(*
Récupère la Config de AppConfig
Démarre HardwareManager
Todo : Démarre la Bdd
Todo : Démarre le monitoring
*)

FUNCTION_BLOCK HardwareControl
VAR_INPUT
END_VAR
VAR_OUTPUT
END_VAR
VAR
	{region "manage file" }	
	{attribute 'OPC.UA.DA' := '0'}	
	_xml : TXml;	
	{attribute 'hide'}
	_filePath : T_MaxString := Const.APP_CONFIG_FILE_PATH; 
	{attribute 'hide'}  			
    _xPath : T_MaxString := Const.APP_CONFIG_XPATH; 
	{endregion}		
		
	{attribute 'hide'}  
	_loadConfigDone : BOOL;
	{attribute 'OPC.UA.DA' := '0'}
	_initialized : BOOL;
	{attribute 'OPC.UA.DA' := '0'}
	_initializedError : BOOL;	
	{attribute 'OPC.UA.DA' := '0'}
	_message : StringBuilder;
	{attribute 'OPC.UA.DA' := '0'}
	_logger : Logger;
	
	autoBoot : BOOL := TRUE;
	
	HardwareManager : HardwareManager;	
END_VAR

IF autoBoot THEN
	InitHardware();
END_IF

ACTION AppDeserialize:
_xml(FilePath := _filePath, XPath := _xPath, 
	 AddHeaderNodeXml := ADR(GlobalConfig.AppConfig), 
	 SizeOfHeaderNodeXml := SIZEOF(GlobalConfig.AppConfig));
END_ACTION

METHOD PRIVATE InitHardware
VAR_INPUT
END_VAR
VAR	
END_VAR
IF _xml.DeserialisationOperation.Ready AND 
   NOT _initialized THEN
    _logger.Information('Initializing hardware...');
END_IF;

IF NOT _initialized  AND NOT _xml.DeserialisationOperation.Error THEN    
	_xml.DeserialisationOperation.Start();
	AppDeserialize();	
END_IF
 
IF _xml.DeserialisationOperation.Done THEN				
	_logger.Debug(_message.Reset().Append('App configuration from ').
						           Append(TO_STRING(Const.APP_CONFIG_FILE_PATH)).ToString());
		
	_logger.Information('App configuration loading done');				
	_xml.DeserialisationOperation.SetReady();
	
	LoadConfigDone := TRUE;	
	_initialized := TRUE;
END_IF
 
IF NOT _initializedError AND _xml.DeserialisationOperation.Error THEN		
	_logger.Error('App configuration loading error');    		
	_xml.SetError(_xml.DeserialisationOperation.ErrorId);
	
	_initializedError := TRUE;
END_IF

IF _loadConfigDone THEN
	HardwareManager();	
END_IF
END_METHOD

PROPERTY LoadConfigDone : BOOL
GET
LoadConfigDone := _loadConfigDone;
END_GET
SET
_loadConfigDone := LoadConfigDone;
END_SET
END_PROPERTY

END_FUNCTION_BLOCK

(* stored: Version 1.1.0.1, ProductVersion 3.1.4024.12
   POU HardwareControl: Id {fa81361c-29a6-4772-bbc9-5971ade645ee}, SpecialFunc None
   Action AppDeserialize: Id {69c1e4cb-6232-4e87-83a9-28a30f5bea14}
   Method InitHardware: Id {e6e410ac-de6a-4ad8-b93a-5d7927e1195b}
   Property LoadConfigDone: Id {f2492bcb-9f94-40ea-9997-a2989502da5e}
   Get Get: Id {76bf09ed-9890-4d51-aee5-b4bd8d01cd82}
   Set Set: Id {d7466f95-34af-454a-a116-819e2e0bb480} *)
